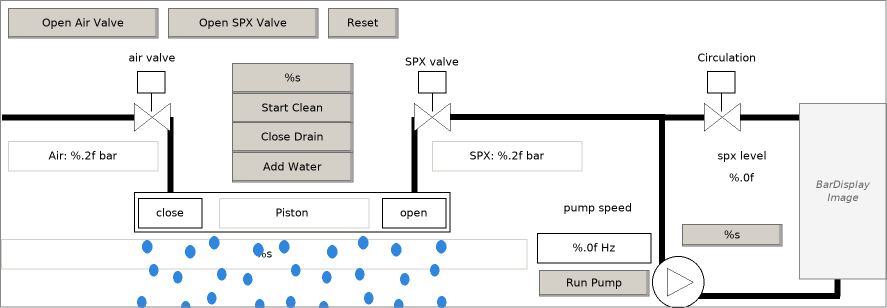
VISUALIZATION visu_Spray  // 887x308
    Button (8,8 150x30), "Open Air Valve", input disabled if: NOT PRG_Spray.bManualActive
        toggle PRG_Spray.bManAirValve p2164770859=TRUE
    Button (539,270 110x26), "Run Pump", input disabled if: NOT PRG_Spray.bManualActive
        toggle PRG_Spray.bManPump p2164770859=TRUE
    Button (168,8 150x30), "Open SPX Valve", input disabled if: NOT PRG_Spray.bManualActive
        toggle PRG_Spray.bManSPXValve
    Button (328,8 70x30), "Reset"
        tap PRG_Spray.bCmdReset
    Polyline (2,117) (134,117)
    Polyline (170,117) (170,200)
    Polyline (414,117) (414,200)
    Polyline (662,117) (704,117)
    Polyline (662,269) (662,117) (450,117)
    Polyline (740,117) (837,117) (837,117)
    Polyline (837,265) (837,296) (690,296)
    Polygon (414,103) (450,131) (450,103) (414,131), colour variable: PRG_Spray.cSPXValve
    Polygon (704,103) (740,131) (740,103) (704,131), colour variable: PRG_Spray.cCircValve
    Line (432,93) (432,111)
    Rectangle (418,71 28x22), colour variable: PRG_Spray.cSPXValve
    Label (102,49 100x18), "air valve"
    Label (357,53 150x18), "SPX valve"
    Label (677,49 100x18), "Circulation"
    Rectangle (537,233 114x30), "%.0f Hz", text variable: GVL_IO.rPumpHzFb
    RoundedRectangle (134,192 316x40)
    Textfield (219,198 150x30), "Piston"
    Rectangle (138,198 64x30), "close", colour variable: PRG_Spray.cPistonClose
    Rectangle (382,198 64x30), "open", colour variable: PRG_Spray.cPistonOpen
    Ellipse (652,256 52x52), colour variable: PRG_Spray.cPump
    Polygon (667,268) (667,296) (693,282)
    Label (523,193 150x30), "pump speed"
    Textfield (704,163 75x30), "%.0f", text variable: GVL_IO.rSPXLevel
        p55702900: PRG_Spray.cLevel
    Line (721,93) (721,111)
    Rectangle (707,71 28x22), colour variable: PRG_Spray.cCircValve
    Line (151,93) (151,111)
    Rectangle (137,71 28x22), colour variable: PRG_Spray.cAirValve
    Polygon (134,103) (170,131) (170,103) (134,131), colour variable: PRG_Spray.cAirValve
    Label (667,141 150x30), "spx level"
    Button (682,224 100x22), "%s", text variable: PRG_Spray.sSimBtnText
        p2175578022: PRG_Spray.cSimBtn
        OnMouseClick: toggle SIM_Plant.bSimEnable
    BarDisplayImage (799,103 88x176), value: GVL_IO.rSPXLevel, style: BarDisplayImage-Green, scale format: %.0f, scale 0..100
    Button (232,63 121x30), "%s", text variable: PRG_Spray.sCleanBtnText, invisible if: NOT PRG_Spray.bManualActive
        toggle PRG_Spray.bBtnClean
    Button (232,93 121x30), "Start Clean", invisible if: NOT PRG_Spray.bCleanActive
        toggle PRG_Spray.bBtnStartClean
    Button (232,122 121x30), "Close Drain", colour toggle: PRG_Spray.bDrainFlash, invisible if: NOT PRG_Spray.bCleanActive
        toggle PRG_Spray.bBtnCloseDrain
    Button (232,152 121x30), "Add Water", colour toggle: PRG_Spray.bWaterFlash, invisible if: NOT PRG_Spray.bCleanActive
        toggle PRG_Spray.bBtnAddWater
    Textfield (1,239 526x30), "%s", text variable: PRG_Spray.sCleanStatus, invisible if: NOT PRG_Spray.bCleanActive
    Textfield (432,141 150x30), "SPX: %.2f bar", text variable: GVL_IO.rSPXPressure
        p55702900: PRG_Spray.cSPXPress
    Textfield (8,141 150x30), "Air: %.2f bar", text variable: GVL_IO.rAirPressure
    Ellipse (142,240 10x13), invisible if: NOT PRG_Spray.abDrop[0]
    Ellipse (185,245 10x13), invisible if: NOT PRG_Spray.abDrop[1]
    Ellipse (209,236 10x13), invisible if: NOT PRG_Spray.abDrop[2]
    Ellipse (253,243 10x13), invisible if: NOT PRG_Spray.abDrop[3]
    Ellipse (279,240 10x13), invisible if: NOT PRG_Spray.abDrop[0]
    Ellipse (327,245 10x13), invisible if: NOT PRG_Spray.abDrop[1]
    Ellipse (358,236 10x13), invisible if: NOT PRG_Spray.abDrop[2]
    Ellipse (391,243 10x13), invisible if: NOT PRG_Spray.abDrop[3]
    Ellipse (436,240 10x13), invisible if: NOT PRG_Spray.abDrop[0]
    Ellipse (149,264 9x12), invisible if: NOT PRG_Spray.abDrop[1]
    Ellipse (173,271 9x12), invisible if: NOT PRG_Spray.abDrop[2]
    Ellipse (217,268 9x12), invisible if: NOT PRG_Spray.abDrop[3]
    Ellipse (243,273 9x12), invisible if: NOT PRG_Spray.abDrop[0]
    Ellipse (291,264 9x12), invisible if: NOT PRG_Spray.abDrop[1]
    Ellipse (322,271 9x12), invisible if: NOT PRG_Spray.abDrop[2]
    Ellipse (355,268 9x12), invisible if: NOT PRG_Spray.abDrop[3]
    Ellipse (400,273 9x12), invisible if: NOT PRG_Spray.abDrop[0]
    Ellipse (430,264 9x12), invisible if: NOT PRG_Spray.abDrop[1]
    Ellipse (137,296 9x12), invisible if: NOT PRG_Spray.abDrop[2]
    Ellipse (181,301 9x12), invisible if: NOT PRG_Spray.abDrop[3]
    Ellipse (207,292 9x12), invisible if: NOT PRG_Spray.abDrop[0]
    Ellipse (255,299 9x12), invisible if: NOT PRG_Spray.abDrop[1]
    Ellipse (286,296 9x12), invisible if: NOT PRG_Spray.abDrop[2]
    Ellipse (319,301 9x12), invisible if: NOT PRG_Spray.abDrop[3]
    Ellipse (364,292 9x12), invisible if: NOT PRG_Spray.abDrop[0]
    Ellipse (394,299 9x12), invisible if: NOT PRG_Spray.abDrop[1]
    Ellipse (437,296 9x12), invisible if: NOT PRG_Spray.abDrop[2]
    Ellipse (145,320 8x11), invisible if: NOT PRG_Spray.abDrop[3]
    Ellipse (171,327 8x11), invisible if: NOT PRG_Spray.abDrop[0]
    Ellipse (219,324 8x11), invisible if: NOT PRG_Spray.abDrop[1]
    Ellipse (250,329 8x11), invisible if: NOT PRG_Spray.abDrop[2]
    Ellipse (283,320 8x11), invisible if: NOT PRG_Spray.abDrop[3]
    Ellipse (328,327 8x11), invisible if: NOT PRG_Spray.abDrop[0]
    Ellipse (358,324 8x11), invisible if: NOT PRG_Spray.abDrop[1]
    Ellipse (401,329 8x11), invisible if: NOT PRG_Spray.abDrop[2]
    Ellipse (425,320 8x11), invisible if: NOT PRG_Spray.abDrop[3]
END_VISUALIZATION

(* stored: Version 1.1.0.1, ProductVersion 3.1.4026.18
   Visu visu_Spray: Id {1f045aa0-71e5-4f9d-bb41-059accc2049b} *)
